TYPE ST_OutputsClosedPalletCheck :
STRUCT
	HW					: ST_HW_OutputsClosedPalletCheck;		
END_STRUCT
END_TYPE

(* stored: Version 1.1.0.1, ProductVersion 3.1.4024.9
   DUT ST_OutputsClosedPalletCheck: Id {e349336d-a962-465d-bbe0-76b39a15ad7c} *)
